TYPE "LaserMarkingBuffer"
VERSION : 0.1
   STRUCT
      DataMatrixStr : String[60];
      ProductNameStr : String[60];
      HW_Str : String[60];
      SW_Str : String[60];
      PN_Str : String[60];
      DATA_Str : String[60];
      SN_Str : String[60];
      ECU_UID_Str : String[60];
      Vdc_Str : String[60];
      Power_Str : String[60];
      Place_Str : String[60];
   END_STRUCT;

END_TYPE

